// TwinCAT 3 PLC project FMRecipes
// Title: FM Recipes
// Company: FrameworkMonorepo
// ProjectVersion: 0.0.1
// ProgramVersion: 3.1.4024.0
// libraries:
//   FM Common Interfaces, * (FrameworkMonorepo)
//   FM Data, * (FrameworkMonorepo)
//   FM Events, * (FrameworkMonorepo)
//   FM Files, * (FrameworkMonorepo)
//   FM Strings, * (FrameworkMonorepo)
//   FM Types, * (FrameworkMonorepo)
//   Tc2_Standard, * (Beckhoff Automation GmbH)
//   Tc2_System, * (Beckhoff Automation GmbH)
//   Tc2_Utilities, * (Beckhoff Automation GmbH)
// project tree:
//   RecipeManager/ RecipeManager.TcPOU, RecipeParameters.TcGVL
//   RecipeManager/RecipeValues/ RecipeAssignment.TcDUT, RecipeSingleValue.TcPOU, RecipeSingleValueType.TcIO, RecipeStringValue.TcPOU, RecipeStringValueType.TcIO, RecipeTableValue.TcPOU, RecipeTableValueType.TcIO, RecipeValue.TcIO
//   Version/ Global_Version.TcGVL
// (motion and I/O tree: see PLC project fmtypes)
// real-time tasks:
//   TASK BindingTestTask: cycle T#1ms, priority 20, ADS port 350
//   TASK PlcTask: cycle T#1ms, priority 21, ADS port 351
//   TASK PlcTask1: cycle T#1ms, priority 22, ADS port 352
//   TASK PlcTask2: cycle T#1ms, priority 23, ADS port 353
//   TASK MathTestTask: cycle T#1ms, priority 24, ADS port 354
//   TASK TimesTestsTask: cycle T#1ms, priority 25, ADS port 355

// ---- RecipeManager/RecipeValues/RecipeAssignment.TcDUT
TYPE RecipeAssignment :
STRUCT
	LineIndex : INT;
	Name : T_MaxString;
	Value : T_MaxString;
	TableRows : INT;
END_STRUCT
END_TYPE

// ---- RecipeManager/RecipeParameters.TcGVL
{attribute 'qualified_only'}
VAR_GLOBAL CONSTANT
	ValueCountLimit : INT := 30;
	TableColumnLimit : INT := 10;
	
	BufferSize : INT := 1500;
	TableBufferSize : INT := 1000;
END_VAR

// ---- Version/Global_Version.TcGVL
{attribute 'TcGenerated'}
{attribute 'no-analysis'}
{attribute 'linkalways'}
// This function has been automatically generated from the project information.
VAR_GLOBAL CONSTANT
	{attribute 'const_non_replaced'}
	stLibVersion_FM_Recipes : ST_LibVersion := (iMajor := 0, iMinor := 0, iBuild := 1, iRevision := 0, nFlags := 0, sVersion := '0.0.1');
END_VAR

// ---- RecipeManager/RecipeValues/RecipeSingleValueType.TcIO
INTERFACE RecipeSingleValueType EXTENDS RecipeValue

METHOD ParseAndAssignValue
VAR_INPUT
	value : T_MaxString;
END_VAR
END_METHOD

END_INTERFACE

// ---- RecipeManager/RecipeValues/RecipeStringValueType.TcIO
INTERFACE RecipeStringValueType EXTENDS RecipeValue

METHOD ParseAndAssignValue
VAR_INPUT
END_VAR
END_METHOD

END_INTERFACE

// ---- RecipeManager/RecipeValues/RecipeTableValueType.TcIO
INTERFACE RecipeTableValueType EXTENDS RecipeValue

METHOD ParseAndAssignValues
VAR_INPUT
	rowCount : INT;
END_VAR
END_METHOD

END_INTERFACE

// ---- RecipeManager/RecipeValues/RecipeValue.TcIO
INTERFACE RecipeValue EXTENDS Disposable

{attribute 'monitoring' := 'call'}
PROPERTY Assignment : STRING
GET
END_GET
SET
END_SET
END_PROPERTY

METHOD BuildAndGetAssignmentString : POINTER TO STRING
END_METHOD

METHOD Dispose
VAR_INPUT
END_VAR
END_METHOD

{attribute 'monitoring' := 'call'}
PROPERTY Name : T_MaxString
GET
END_GET
SET
END_SET
END_PROPERTY

END_INTERFACE

// ---- RecipeManager/RecipeManager.TcPOU
FUNCTION_BLOCK RecipeManager IMPLEMENTS Cyclic, Name
VAR
	values : ARRAY[0..RecipeParameters.ValueCountLimit - 1] OF RecipeValue;
	valueCount : INT;

	valueStringBuffer : STRING(RecipeParameters.TableBufferSize);
	_Buffer : STRING(RecipeParameters.BufferSize);
	sb : StringBuilderExtBuffer := (Buffer := ToAnyType(_Buffer));

	_FolderPath : T_MaxString;
	_FileName : T_MaxString;
	file : File;
	savingFile : BOOL;
	loadingFile : BOOL;
	directory : Directory;
	
	_JustLoaded : BOOL;
	_JustSaved : BOOL;

	_NewLine : STRING := '$N';
	_Assignment : STRING := ':=';
	_Extension : STRING := '.txt';
	_StringBoundary : STRING := '$'';
	
	_Name : T_MaxString;
	
	savedMessage : MessageEventLogger(TC_EVENTS.RecipeManagerEventClass.RecipeManagerSavedRecipe) := (Source := THIS^);
	loadedMessage : MessageEventLogger(TC_EVENTS.RecipeManagerEventClass.RecipeManagerLoadedRecipe) := (Source := THIS^);
END_VAR

METHOD AddSingleValue
VAR_INPUT
	value : ANY;
	name : T_MaxString;
END_VAR
VAR
	newValue : POINTER TO RecipeSingleValue;
END_VAR
IF (valueCount < RecipeParameters.ValueCountLimit) THEN
	newValue := __NEW(RecipeSingleValue);
	newValue^.Bind(value);
	newValue^.Name := name;
	newValue^.Assignment := _Assignment;
	values[valueCount] := newValue^;
	
	valueCount := valueCount + 1;
END_IF
END_METHOD

METHOD AddStringValue
VAR_INPUT
	value : ANY;
	name : T_MaxString;
END_VAR
VAR
	newValue : POINTER TO RecipeStringValue;
END_VAR
IF (valueCount < RecipeParameters.ValueCountLimit) THEN
	newValue := __NEW(RecipeStringValue);
	newValue^.Bind(value);
	newValue^.Buffer := ToAnyType(valueStringBuffer);
	newValue^.Name := name;
	newValue^.Assignment := _Assignment;
	values[valueCount] := newValue^;
	
	valueCount := valueCount + 1;
END_IF
END_METHOD

METHOD AddTableValue : REFERENCE TO RecipeTableValue
VAR_INPUT
	firstRow : ANY;
	name : T_MaxString;
END_VAR
VAR
	newValue : POINTER TO RecipeTableValue;
END_VAR
IF (valueCount < RecipeParameters.ValueCountLimit) THEN
	newValue := __NEW(RecipeTableValue);
	newValue^.Buffer := ToAnyType(valueStringBuffer);
	newValue^.DefineRow(firstRow);
	newValue^.Name := name;
	newValue^.Assignment := _Assignment;
	values[valueCount] := newValue^;
	
	valueCount := valueCount + 1;
	
	AddTableValue REF= newValue^;
END_IF
END_METHOD

{attribute 'monitoring' := 'call'}
PROPERTY Assignment : STRING
GET
Assignment := _Assignment;
END_GET
SET
_Assignment := Assignment;
END_SET
END_PROPERTY

PROPERTY BuildParseBuffer : REFERENCE TO StringBuilderExtBuffer
GET
BuildParseBuffer REF= sb;
END_GET
END_PROPERTY

METHOD BuildValueString : BOOL
VAR
	i : INT;
END_VAR
sb.Clear();
FOR i := 0 TO valueCount - 1 DO
	IF (i > 0) THEN
		sb.Append(_NewLine);
	END_IF
	sb.AppendByPointer(values[i].BuildAndGetAssignmentString());
END_FOR
END_METHOD

{attribute 'monitoring' := 'call'}
PROPERTY Busy : BOOL
GET
Busy := savingFile OR loadingFile;
END_GET
END_PROPERTY

METHOD Cyclic
file.Cyclic();
directory.Cyclic();

_JustSaved := FALSE;
_JustLoaded := FALSE;

IF (savingFile AND file.Done) THEN
	savingFile := FALSE;
	_JustSaved := TRUE;
	sb.Clear();
	ListRecipes();
	savedMessage.ClearArguments().AddStringByValue(_FileName);
	savedMessage.Send();
END_IF

IF (loadingFile AND file.Done) THEN
	loadingFile := FALSE;
	_JustLoaded := TRUE;
	ParseValueString();
	sb.Clear();
	loadedMessage.ClearArguments().AddStringByValue(_FileName);
	loadedMessage.Send();
END_IF

IF (NOT directory.ListDone) THEN
	ListRecipes();
END_IF
END_METHOD

{attribute 'monitoring' := 'call'}
PROPERTY Extension : STRING
GET
Extension := _Extension;
END_GET
SET
_Extension := Extension;
END_SET
END_PROPERTY

METHOD FB_exit : BOOL
VAR_INPUT
	bInCopyCode : BOOL; // if TRUE, the exit method is called for exiting an instance that is copied afterwards (online change).
END_VAR
VAR
	i : INT;
END_VAR
FOR i := 0 TO valueCount - 1 DO
	values[i].Dispose();
	values[i] := 0;
END_FOR
END_METHOD

METHOD FB_init : BOOL
VAR_INPUT
	bInitRetains : BOOL; // if TRUE, the retain variables are initialized (warm start / cold start)
	bInCopyCode : BOOL;  // if TRUE, the instance afterwards gets moved into the copy code (online change)
END_VAR
END_METHOD

{attribute 'monitoring' := 'call'}
PROPERTY FileName : T_MaxString
GET
FileName := _FileName;
END_GET
SET
_FileName := FileName;
END_SET
END_PROPERTY

{attribute 'monitoring' := 'call'}
PROPERTY FolderPath : T_MaxString
GET
FolderPath := _FolderPath;
END_GET
SET
_FolderPath := FolderPath;
END_SET
END_PROPERTY

METHOD PRIVATE GetRecipePath : T_MaxString
GetRecipePath := CONCAT(_FolderPath, _FileName);

IF (NOT StringEndsWithAny(_FileName, _Extension)) THEN
	GetRecipePath := CONCAT(GetRecipePath, _Extension);
END_IF
END_METHOD

METHOD GetTable : REFERENCE TO RecipeTableValue
VAR_INPUT
	name : T_MaxString;
END_VAR
VAR
	value : RecipeValue;
	p : POINTER TO RecipeTableValue;
END_VAR
value := GetValue(name);
__QUERYPOINTER(value, p);
IF (p <> 0) THEN
	GetTable REF= p^;
END_IF
END_METHOD

METHOD GetValue : RecipeValue
VAR_INPUT
	name : T_MaxString;
END_VAR
VAR
	i : INT;
END_VAR
FOR i := 0 TO valueCount - 1 DO
	IF (values[i].Name = name) THEN
		GetValue := values[i];
		RETURN;
	END_IF
END_FOR
END_METHOD

{attribute 'monitoring' := 'call'}
PROPERTY JustLoaded : BOOL
GET
JustLoaded := _JustLoaded;
END_GET
END_PROPERTY

{attribute 'monitoring' := 'call'}
PROPERTY JustSaved : BOOL
GET
JustSaved := _JustSaved;
END_GET
END_PROPERTY

{attribute 'monitoring' := 'call'}
PROPERTY ListLoaded : BOOL
GET
ListLoaded := directory.ListDone;
END_GET
END_PROPERTY

METHOD ListRecipes
VAR_INPUT
END_VAR
directory.List(
	BuildStringInline(_FolderPath)
		.Append('*')
		.Append(_Extension)
		.GetString()
);
END_METHOD

METHOD Load
IF (_FileName = '' OR _FolderPath = '') THEN
	RETURN;
END_IF

sb.Clear();

file.Read(
	buffer := ADR(_Buffer),
	bufferLength := SIZEOF(_Buffer) - 1,
	filePath := GetRecipePath()
);

loadingFile := TRUE;
END_METHOD

{attribute 'monitoring' := 'call'}
PROPERTY Name : T_MaxString
GET
Name := _Name;
END_GET
SET
_Name := Name;
END_SET
END_PROPERTY

{attribute 'monitoring' := 'call'}
PROPERTY NewLine : STRING
GET
NewLine := _NewLine;
END_GET
SET
_NewLine := NewLine;

//serializer.NewLine := _NewLine;
//deserializer.NewLine := _NewLine;
END_SET
END_PROPERTY

METHOD PRIVATE ParseValueString
VAR
	caret : DINT;
	assignmentLength : DINT;
	newLineLength : DINT;
	variableNameLength : DINT;
	variableName : T_MaxString;
	tableRowCountString : STRING;
	tableRowCount : INT;
	singleValueString : T_MaxString;
	valueLength : DINT;
	tableLineLength : DINT;
	newLineIndex : DINT;
	stringBoundaryLength : DINT;
	
	value : RecipeValue;
	singleValue : RecipeSingleValueType;
	stringValue : RecipeStringValueType;
	tableValue : RecipeTableValueType;
	
	sbValueBuffer : StringBuilderExtBuffer := (Buffer := ToAnyType(valueStringBuffer));

	i : INT;
END_VAR
sb.UpdateBufferLength();

assignmentLength := LEN(_Assignment);
newLineLength := LEN(_NewLine);
stringBoundaryLength := LEN(_StringBoundary);
WHILE caret < sb.Length DO
	// Search for assignment string
	variableNameLength := TO_DINT(FIND2(ADR(_Buffer[caret]), ADR(_Assignment))) - 1;
	IF (variableNameLength <= 0 OR variableNameLength > SIZEOF(T_MaxString) - 1) THEN
		EXIT;
	END_IF
	
	// Get variable name
	ClearData(variableName);
	SubString(_Buffer, variableName, caret, variableNameLength);
	variableName := F_LTrim(F_RTrim(variableName));
	tableRowCountString := F_LTrim(F_RTrim(GetStringBetween(variableName, '[', ']')));
	IF (LEN(tableRowCountString) > 0) THEN
		tableRowCount := STRING_TO_INT(tableRowCountString);
		variableName := LEFT(variableName, LEN(variableName) - LEN(tableRowCountString) - 2);
	ELSE
		tableRowCount := 0;
	END_IF
	
	caret := caret + variableNameLength + assignmentLength;
	
	// Find value by name
	value := GetValue(variableName);
	IF (value = 0) THEN
		CONTINUE;
	END_IF
	
	// Get value string
	// Parse and assign value
	// Update caret
	ClearData(singleValueString);
	IF (__QUERYINTERFACE(value, singleValue)) THEN
		valueLength := TO_DINT(FIND2(pSrcString := ADR(_Buffer[caret]), pFindString := ADR(_NewLine))) - 1;
		IF (valueLength < 0) THEN
			valueLength := sb.Length - caret;
		ELSIF (valueLength > SIZEOF(T_MaxString) - 1) THEN
			EXIT;
		END_IF
		SubString(_Buffer, singleValueString, caret, valueLength);
		singleValueString := F_LTrim(F_RTrim(singleValueString));
		singleValue.ParseAndAssignValue(singleValueString);
		caret := caret + valueLength + newLineLength;
	ELSIF (__QUERYINTERFACE(value, stringValue)) THEN
		caret := caret + TO_DINT(FIND2(
								pSrcString := ADR(_Buffer[caret]),
								pFindString := ADR(_StringBoundary)
						)) - 1 + stringBoundaryLength;
		valueLength := 0;
		WHILE TRUE DO
			valueLength := valueLength + TO_DINT(FIND2(
											pSrcString := ADR(_Buffer[caret + valueLength]),
											pFindString := ADR(_StringBoundary))
										) - 1;
			IF (valueLength = -1) THEN
				EXIT;
			ELSIF (caret + valueLength + 2 * stringBoundaryLength < sb.Length) THEN
				IF (StringBeginsWith(PSTRING_TO_STRING(ADR(_Buffer) + TO_DWORD(caret + valueLength + stringBoundaryLength)), _StringBoundary)) THEN
					valueLength := valueLength + 2 * stringBoundaryLength;
				ELSE 
					EXIT;
				END_IF 
			ELSE
				EXIT;
			END_IF
		END_WHILE
		sbValueBuffer.Clear().AppendSubString(_Buffer, caret, valueLength);
		stringValue.ParseAndAssignValue();
		newLineIndex := TO_DINT(FIND2(
									pSrcString := ADR(_Buffer[caret + valueLength + stringBoundaryLength]),
									pFindString := ADR(_NewLine)
							)) - 1;
		caret := caret + valueLength + stringBoundaryLength + newLineIndex + newLineLength;
	ELSIF (__QUERYINTERFACE(value, tableValue)) THEN
		FOR i := 0 TO 1 DO
			caret := caret + TO_DINT(FIND2(
									pSrcString := ADR(_Buffer[caret]),
									pFindString := ADR(_NewLine)
							)) - 1 + newLineLength;
		END_FOR
		valueLength := 0;
		FOR i := 0 TO tableRowCount - 1 DO
			tableLineLength := TO_DINT(FIND2(
									pSrcString := ADR(_Buffer[caret + valueLength]),
									pFindString := ADR(_NewLine)
							)) - 1 + newLineLength;
			IF (tableLineLength = 0) THEN
				tableLineLength := sb.Length - (caret + valueLength);
			END_IF
			valueLength := valueLength + tableLineLength;
		END_FOR
		sbValueBuffer.Clear().AppendSubString(_Buffer, caret, valueLength);
		tableValue.ParseAndAssignValues(tableRowCount);
		caret := caret + valueLength; // Newline is already included in table row search
	END_IF
END_WHILE
END_METHOD

METHOD RecipeExists : BOOL
VAR_INPUT
	name : T_MaxString;
END_VAR
VAR
	fileName : T_MaxString;
	i : INT;
	list : REFERENCE TO ARRAY[0..49] OF T_MaxString;
END_VAR
IF (name = '') THEN
	RETURN;
END_IF

IF (StringEndsWithAny(name, _Extension)) THEN
	fileName := name;
ELSE
	fileName := CONCAT(name, _Extension);
END_IF

list REF= RecipeList;
FOR i := 0 TO 49 DO
	IF (list[i] = '') THEN
		RETURN;
	END_IF
	IF (list[i] = fileName) THEN
		RecipeExists := TRUE;
		RETURN;
	END_IF
END_FOR
END_METHOD

{attribute 'monitoring' := 'call'}
PROPERTY RecipeList : REFERENCE TO ARRAY[0..49] OF T_MaxString
GET
RecipeList REF= directory.FileNameList;
END_GET
END_PROPERTY

METHOD Save
IF (_FileName = '' OR _FolderPath = '') THEN
	RETURN;
END_IF

BuildValueString();

file.Write(
	buffer := ADR(_Buffer),
	bufferLength := LEN2(ADR(_Buffer)),
	filePath := GetRecipePath(),
	append := FALSE
);

savingFile := TRUE;
END_METHOD

END_FUNCTION_BLOCK

// ---- RecipeManager/RecipeValues/RecipeSingleValue.TcPOU
{attribute 'enable_dynamic_creation'}
FUNCTION_BLOCK RecipeSingleValue IMPLEMENTS RecipeSingleValueType
VAR
	_Name : T_MaxString;
	_Value : __SYSTEM.AnyType;
	_Assignment : STRING := ':=';
	_AssignmentString : T_MaxString;
END_VAR

{attribute 'monitoring' := 'call'}
PROPERTY Assignment : STRING
GET
Assignment := _Assignment;
END_GET
SET
_Assignment := Assignment;
END_SET
END_PROPERTY

METHOD Bind
VAR_INPUT
	value : ANY;
END_VAR
_Value := value;
END_METHOD

METHOD BuildAndGetAssignmentString : POINTER TO STRING
VAR_INPUT
END_VAR
_AssignmentString := 
	BuildStringInline(_Name)
	.Append(_Assignment)
	.Append(ValueString)
	.GetString();
BuildAndGetAssignmentString := ADR(_AssignmentString);
END_METHOD

METHOD Dispose
VAR_INPUT
END_VAR
__DELETE(THIS);
END_METHOD

{attribute 'monitoring' := 'call'}
PROPERTY Name : T_MaxString
GET
Name := _Name;
END_GET
SET
_Name := Name;
END_SET
END_PROPERTY

METHOD ParseAndAssignValue
VAR_INPUT
	value : T_MaxString;
END_VAR
StringToAnyType(value, _Value);
END_METHOD

{attribute 'monitoring' := 'call'}
PROPERTY ValueString : T_MaxString
GET
IF (IsAnyTypeBound(_Value)) THEN
	ValueString := AnyTypeToString(_Value);
END_IF
END_GET
END_PROPERTY

END_FUNCTION_BLOCK

// ---- RecipeManager/RecipeValues/RecipeStringValue.TcPOU
{attribute 'enable_dynamic_creation'}
FUNCTION_BLOCK RecipeStringValue IMPLEMENTS RecipeStringValueType
VAR
	_Name : T_MaxString;
	_Value : __SYSTEM.AnyType;
	_Assignment : STRING := ':=';
	_StringBoundary : STRING := '$'';
	
	sb : StringBuilderExtBuffer;
END_VAR

{attribute 'monitoring' := 'call'}
PROPERTY Assignment : STRING
GET
Assignment := _Assignment;
END_GET
SET
_Assignment := Assignment;
END_SET
END_PROPERTY

METHOD Bind
VAR_INPUT
	value : ANY;
END_VAR
_Value := value;
END_METHOD

PROPERTY Buffer : __SYSTEM.AnyType
GET
Buffer := sb.Buffer;
END_GET
SET
sb.Buffer := Buffer;
END_SET
END_PROPERTY

METHOD BuildAndGetAssignmentString : POINTER TO STRING
VAR
	anyToWrite : __SYSTEM.AnyType;
END_VAR
sb.Clear();
sb.Append(
	BuildStringInline(_Name)
	.Append(_Assignment)
	.Append(_StringBoundary)
	.GetString()
);

anyToWrite.pValue := __NEW(BYTE, TO_UDINT(_Value.diSize));
anyToWrite.diSize := _Value.diSize;
MEMSET(anyToWrite.pValue, 0, TO_UDINT(_Value.diSize));
MEMCPY(anyToWrite.pValue, _Value.pValue, TO_UDINT(_Value.diSize));
ReplaceAllAnyType(anyToWrite, _StringBoundary, CONCAT(_StringBoundary, _StringBoundary));

sb.AppendByPointer(anyToWrite.pValue);
__DELETE(anyToWrite.pValue);

sb.Append(_StringBoundary);
BuildAndGetAssignmentString := sb.BufferRef.pValue;
END_METHOD

METHOD Dispose
VAR_INPUT
END_VAR
__DELETE(THIS);
END_METHOD

{attribute 'monitoring' := 'call'}
PROPERTY Name : T_MaxString
GET
Name := _Name;
END_GET
SET
_Name := Name;
END_SET
END_PROPERTY

METHOD ParseAndAssignValue
VAR_INPUT
END_VAR
ClearDataAnyType(_Value);
ReplaceAllAnyType(sb.BufferRef, CONCAT(_StringBoundary, _StringBoundary), _StringBoundary);
MEMCPY(
	destAddr := _Value.pValue,
	srcAddr := sb.BufferRef.pValue,
	n := MIN(DINT_TO_UDINT(_Value.diSize - 1), LEN2(sb.BufferRef.pValue))
);
END_METHOD

{attribute 'monitoring' := 'call'}
PROPERTY ValueString : T_MaxString
GET
IF (IsAnyTypeBound(_Value)) THEN
	ValueString := AnyTypeToString(_Value);
END_IF
END_GET
END_PROPERTY

END_FUNCTION_BLOCK

// ---- RecipeManager/RecipeValues/RecipeTableValue.TcPOU
{attribute 'enable_dynamic_creation'}
FUNCTION_BLOCK RecipeTableValue IMPLEMENTS RecipeTableValueType
VAR
	_Name : T_MaxString;
	_Table : __SYSTEM.AnyType;
	_ColumnNames : ARRAY[0..RecipeParameters.TableColumnLimit - 1] OF T_MaxString;
	_ColumnDefinitions : ARRAY[0..RecipeParameters.TableColumnLimit - 1] OF __SYSTEM.AnyType;
	_Assignment : STRING := ':=';
	_NewLine : STRING := '$N';
	
	sb : StringBuilderExtBuffer;
	serializer : TableSerializer := (
		Stringbuilder := sb
	);
	deserializer : TableDeserializer;
END_VAR

{attribute 'monitoring' := 'call'}
PROPERTY Assignment : STRING
GET
Assignment := _Assignment;
END_GET
SET
_Assignment := Assignment;
END_SET
END_PROPERTY

PROPERTY Buffer : __SYSTEM.AnyType
GET
Buffer := sb.Buffer;
END_GET
SET
sb.Buffer := Buffer;
deserializer.DataString := Buffer.pValue;
END_SET
END_PROPERTY

METHOD BuildAndGetAssignmentString : POINTER TO STRING
VAR_INPUT
END_VAR
sb.Clear();
sb.Append(
	BuildStringInline(_Name)
	.Append('[')
	.Append(TO_STRING(serializer.RowCount))
	.Append('] ')
	.Append(_Assignment)
	.Append(_Newline)
	.GetString()
);
serializer.Serialize(TRUE, FALSE);
BuildAndGetAssignmentString := sb.BufferRef.pValue;
END_METHOD

METHOD DefineNextColumn : REFERENCE TO RecipeTableValue
VAR_INPUT
	columnInFirstRow : ANY;
	name : T_MaxString;
END_VAR
serializer.DefineNextColumnWithName(columnInFirstRow, name);
deserializer.DefineNextColumn(columnInFirstRow);

DefineNextColumn REF= THIS^;
END_METHOD

METHOD DefineRow : REFERENCE TO RecipeTableValue
VAR_INPUT
	firstRow : ANY;
END_VAR
serializer.DefineRow(firstRow);
deserializer.DefineRow(firstRow);

DefineRow REF= THIS^;
END_METHOD

METHOD Dispose
VAR_INPUT
END_VAR
__DELETE(THIS);
END_METHOD

{attribute 'monitoring' := 'call'}
PROPERTY Name : T_MaxString
GET
Name := _Name;
END_GET
SET
_Name := Name;
END_SET
END_PROPERTY

{attribute 'monitoring' := 'call'}
PROPERTY NewLine : STRING
GET
NewLine := _NewLine;
END_GET
SET
_NewLine := NewLine;

serializer.NewLine := _NewLine;
deserializer.NewLine := _NewLine;
END_SET
END_PROPERTY

METHOD ParseAndAssignValues
VAR_INPUT
	rowCount : INT;
END_VAR
VAR
END_VAR
THIS^.RowCount := rowCount;
deserializer.Deserialize(FALSE);
END_METHOD

{attribute 'monitoring' := 'call'}
PROPERTY RowCount : DINT
GET
RowCount := serializer.RowCount;
END_GET
SET
serializer.RowCount := RowCount;
deserializer.RowCount := RowCount;
END_SET
END_PROPERTY

END_FUNCTION_BLOCK
